% RSLogix 500 project SW2012_BE.RSS, saved by version 12.00.00.00 %
PROJECT "PS8"    % processor: MicroLogix 1400 %

PROGRAM FILES
  LAD 2 "MAIN"  23 rungs  % Calls all system and subsystem routines %
  LAD 3 "CONSTANTS"  50 rungs  % Maintains the system constants %
  LAD 4 "DEFAULTS"  54 rungs  % Manages the system default values %
  LAD 5 "SYS_FAULTS"  45 rungs  % Monitors the system fault conditions %
  LAD 6 "SYSTEM"  71 rungs  % Controls the system %
  LAD 7 "PROCESSING"  17 rungs  % Runs the processing control %
  LAD 8 "MANUAL_CTL"  9 rungs  % Runs the manual valve control %
  LAD 10 "PURIFY"  37 rungs  % Operates the purify control %
  LAD 11 "REGEN"  79 rungs  % Operates the regen control %
  LAD 12 "REGEN_FLT"  47 rungs  % regen alarms and warnings %
  LAD 17 "BYPASS"  7 rungs  % Controls the bypass %
  LAD 18 "MIX PANEL"  12 rungs
  LAD 20 "ADS_A"  47 rungs  % Controls the Adsorber A %
  LAD 21 "ADS_A_FLT"  17 rungs  % Controls the Adsorber A faults %
  LAD 22 "ADS_B"  47 rungs  % Controld Adsorber B %
  LAD 23 "ADS_B_FLT"  17 rungs  % Controls the Adsorber B faults %
  LAD 24 "PREHEATER"  9 rungs
  LAD 25 "PH_FLT"  15 rungs
  LAD 49 "MODBUS"  37 rungs
  LAD 50 "PLC_FAULT"  2 rungs
  LAD 51 "REVERSE"  9 rungs

DATA FILES
  O0 OUTPUT  24 elements
  I1 INPUT  25 elements
  S2 STATUS  66 elements
  B3 BINARY  4 elements
  T4 TIMER  112 elements
  C5 COUNTER  21 elements
  R6 CONTROL  2 elements
  N7 SYSTEM CFG  120 elements  % Maintains the values that characterize the system %
  F8 FLOAT  3 elements
  N9 CONSTANTS  86 elements  % The collection of system and subsystem constants %
  N10 SYSTEM  30 elements  % Contain the values for system control %
  N11 PROCESS  4 elements  % Contains the values for the processing machine %
  N12 PURIFY  25 elements  % Contains the values required for purify %
  N13 REGEN  31 elements  % Contains the values required for regen %
  N15 MANUAL CTL  5 elements  % Contains the data for the manual valve control %
  N16 ADSORBER_A  22 elements  % Contains the values for Adsorber A %
  N17 ADSORBER_B  22 elements  % Contains the values required for Adsorber B %
  N19 BYPASS  2 elements
  N20 MIX PANEL  7 elements
  N21 NOMEMBCKUP  4 elements
  PD25 PID HEATER  4 elements
  B30 SYSTEM CFG  6 elements
  B31 SYSTEM  18 elements
  B32 PROCESS  1 elements
  B33 PURIFY  2 elements
  B34 REGEN  3 elements
  B35 MANUAL CTL  3 elements
  B38 BYPASS  1 elements
  L52 SERIAL  1 elements
  N64 MODBUS  126 elements
  L65 TOTAL FLOW  1 elements
  MG68   1 elements
  B69   3 elements
  RIX80   1 elements
  N200 STATUS_SYS  1 elements  % HMI System Status %
  L201 STATUS_PUR  1 elements  % HMI Purifier Status  %
  L202 STATUS_GET  3 elements  % HMI Getter Status %
  L203 STATUS_ADS  3 elements  % HMI Adsorber Status %
  F206 FLOAT_PRC  4 elements  % HMI Purify function Float Values %
  N207 STATUS_PRC  7 elements  % HMI Purify Process function status %
  N210 BUZZER  5 elements  % ALARM BUZZER CONTROL %

LADDER 2 "MAIN"    % Calls all system and subsystem routines %
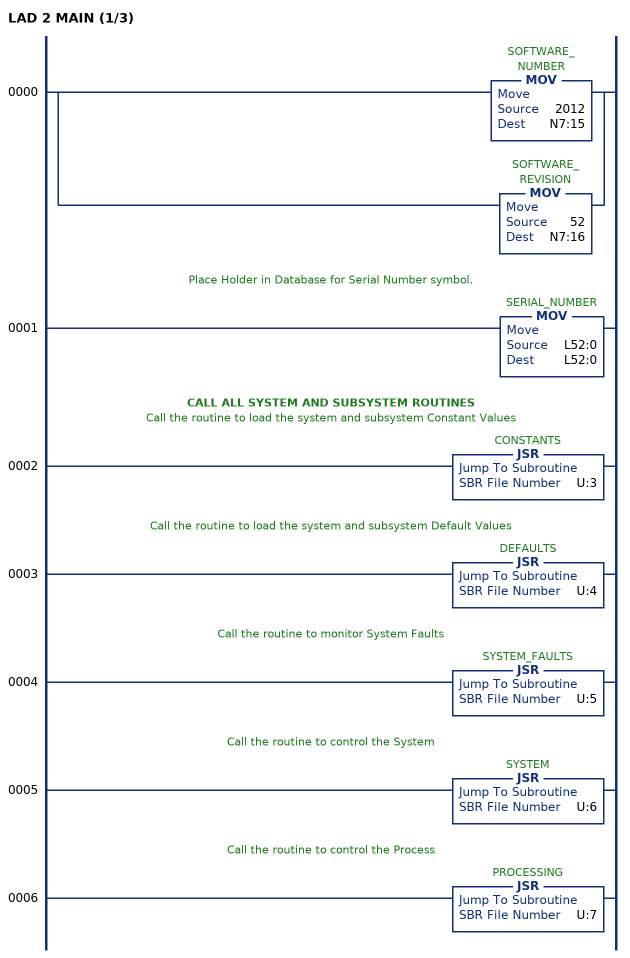
% Rung: 0 %
SOR BST MOV 2012 N7:15 NXB MOV 52 N7:16 BND EOR
%   N7:15  SOFTWARE_NUMBER %
%   N7:16  SOFTWARE_REVISION %
% Rung: 1 %
% Place Holder in Database for Serial Number symbol. %
SOR MOV L52:0 L52:0 EOR
%   L52:0  SERIAL_NUMBER %
% Rung: 2 %
% TITLE: CALL ALL SYSTEM AND SUBSYSTEM ROUTINES %
% Call the routine to load the system and subsystem Constant Values %
SOR JSR U:3 EOR
%   U:3  CONSTANTS %
% Rung: 3 %
% Call the routine to load the system and subsystem Default Values %
SOR JSR U:4 EOR
%   U:4  DEFAULTS %
% Rung: 4 %
% Call the routine to monitor System Faults %
SOR JSR U:5 EOR
%   U:5  SYSTEM_FAULTS %
% Rung: 5 %
% Call the routine to control the System %
SOR JSR U:6 EOR
%   U:6  SYSTEM %
% Rung: 6 %
% Call the routine to control the Process %
SOR JSR U:7 EOR
%   U:7  PROCESSING %

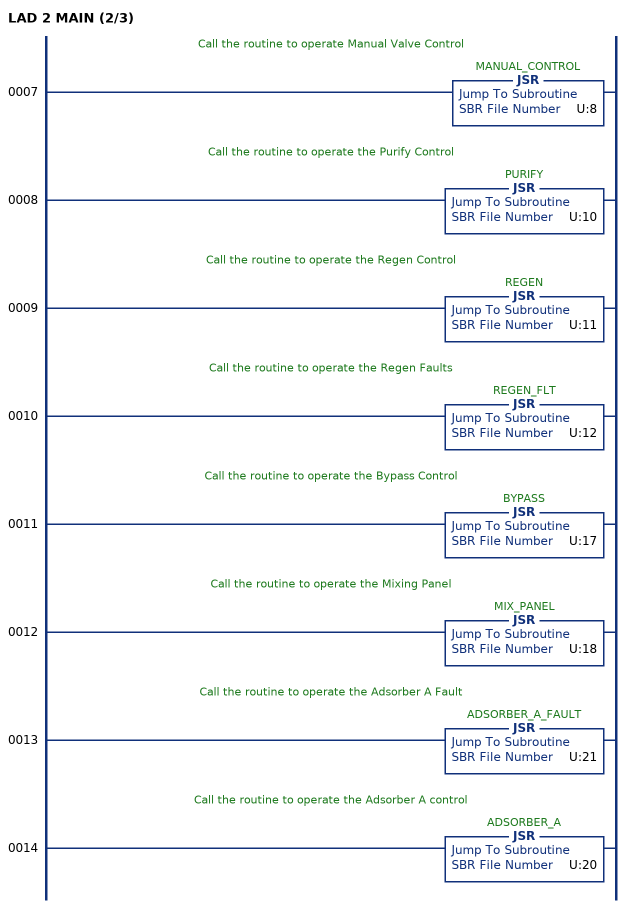
% Rung: 7 %
% Call the routine to operate Manual Valve Control %
SOR JSR U:8 EOR
%   U:8  MANUAL_CONTROL %
% Rung: 8 %
% Call the routine to operate the Purify Control %
SOR JSR U:10 EOR
%   U:10  PURIFY %
% Rung: 9 %
% Call the routine to operate the Regen Control %
SOR JSR U:11 EOR
%   U:11  REGEN %
% Rung: 10 %
% Call the routine to operate the Regen Faults %
SOR JSR U:12 EOR
%   U:12  REGEN_FLT %
% Rung: 11 %
% Call the routine to operate the Bypass Control %
SOR JSR U:17 EOR
%   U:17  BYPASS %
% Rung: 12 %
% Call the routine to operate the Mixing Panel %
SOR JSR U:18 EOR
%   U:18  MIX_PANEL %
% Rung: 13 %
% Call the routine to operate the Adsorber A Fault %
SOR JSR U:21 EOR
%   U:21  ADSORBER_A_FAULT %
% Rung: 14 %
% Call the routine to operate the Adsorber A control %
SOR JSR U:20 EOR
%   U:20  ADSORBER_A %

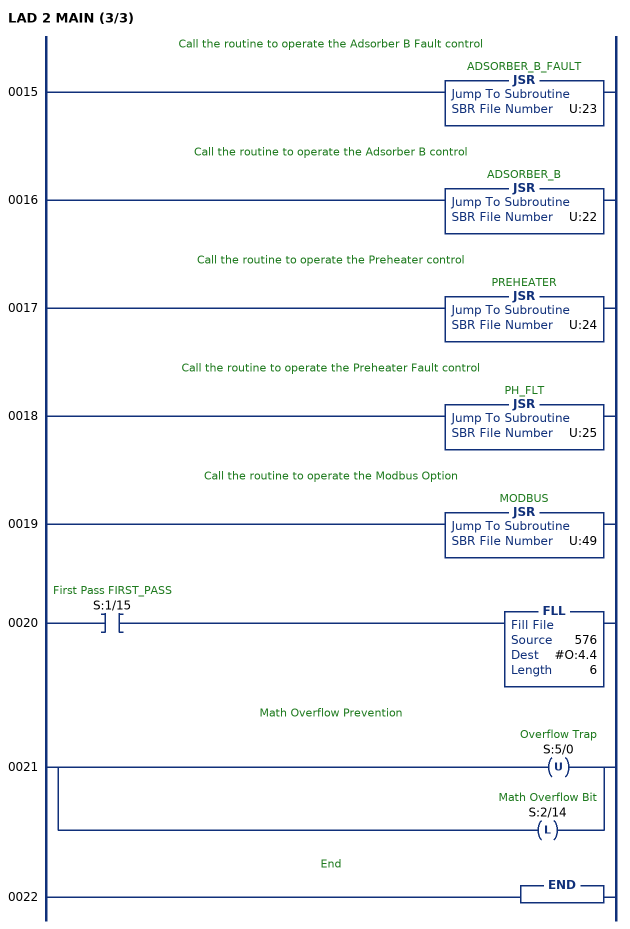
% Rung: 15 %
% Call the routine to operate the Adsorber B Fault control %
SOR JSR U:23 EOR
%   U:23  ADSORBER_B_FAULT %
% Rung: 16 %
% Call the routine to operate the Adsorber B control %
SOR JSR U:22 EOR
%   U:22  ADSORBER_B %
% Rung: 17 %
% Call the routine to operate the Preheater control %
SOR JSR U:24 EOR
%   U:24  PREHEATER %
% Rung: 18 %
% Call the routine to operate the Preheater Fault control %
SOR JSR U:25 EOR
%   U:25  PH_FLT %
% Rung: 19 %
% Call the routine to operate the Modbus Option %
SOR JSR U:49 EOR
%   U:49  MODBUS %
% Rung: 20 %
SOR XIC S:1/15 FLL 576 #O:4.4 6 EOR
%   S:1/15  FIRST_PASS  "First Pass" %
% Rung: 21 %
% Math Overflow Prevention %
SOR BST OTU S:5/0 NXB OTL S:2/14 BND EOR
%   S:5/0  "Overflow Trap" %
%   S:2/14  "Math Overflow Bit" %
% Rung: 22 %
% End %
SOR END EOR

LADDER 3 "CONSTANTS"    % Maintains the system constants %
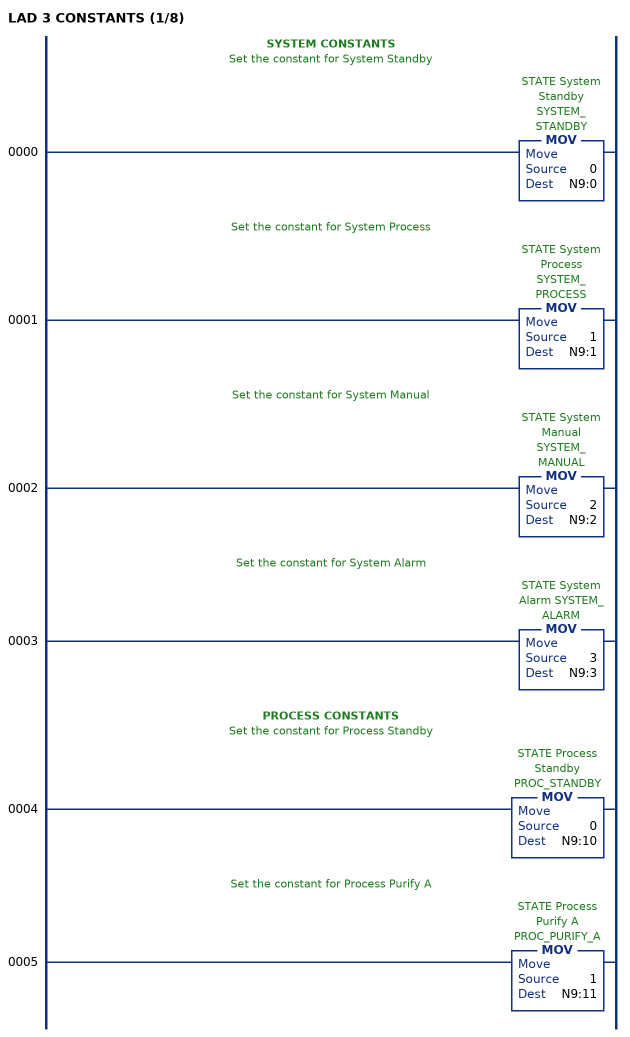
% Rung: 0 %
% TITLE: SYSTEM CONSTANTS %
% Set the constant for System Standby %
SOR MOV 0 N9:0 EOR
%   N9:0  SYSTEM_STANDBY  "STATE System Standby" %
% Rung: 1 %
% Set the constant for System Process %
SOR MOV 1 N9:1 EOR
%   N9:1  SYSTEM_PROCESS  "STATE System Process" %
% Rung: 2 %
% Set the constant for System Manual %
SOR MOV 2 N9:2 EOR
%   N9:2  SYSTEM_MANUAL  "STATE System Manual" %
% Rung: 3 %
% Set the constant for System Alarm %
SOR MOV 3 N9:3 EOR
%   N9:3  SYSTEM_ALARM  "STATE System Alarm" %
% Rung: 4 %
% TITLE: PROCESS CONSTANTS %
% Set the constant for Process Standby %
SOR MOV 0 N9:10 EOR
%   N9:10  PROC_STANDBY  "STATE Process Standby" %
% Rung: 5 %
% Set the constant for Process Purify A %
SOR MOV 1 N9:11 EOR
%   N9:11  PROC_PURIFY_A  "STATE Process Purify A" %

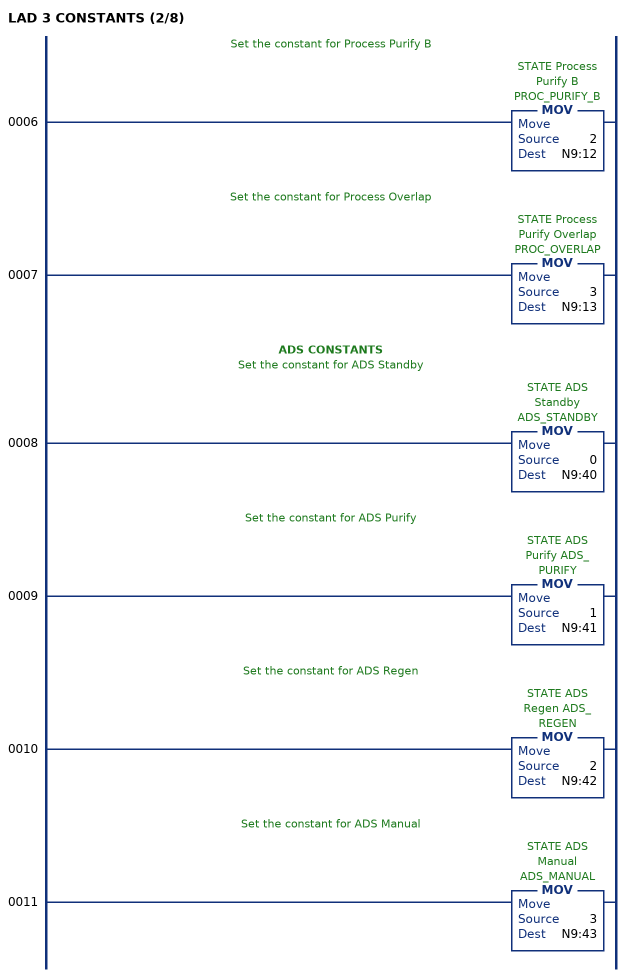
% Rung: 6 %
% Set the constant for Process Purify B %
SOR MOV 2 N9:12 EOR
%   N9:12  PROC_PURIFY_B  "STATE Process Purify B" %
% Rung: 7 %
% Set the constant for Process Overlap %
SOR MOV 3 N9:13 EOR
%   N9:13  PROC_OVERLAP  "STATE Process Purify Overlap" %
% Rung: 8 %
% TITLE: ADS CONSTANTS %
% Set the constant for ADS Standby %
SOR MOV 0 N9:40 EOR
%   N9:40  ADS_STANDBY  "STATE ADS Standby" %
% Rung: 9 %
% Set the constant for ADS Purify %
SOR MOV 1 N9:41 EOR
%   N9:41  ADS_PURIFY  "STATE ADS Purify" %
% Rung: 10 %
% Set the constant for ADS Regen %
SOR MOV 2 N9:42 EOR
%   N9:42  ADS_REGEN  "STATE ADS Regen" %
% Rung: 11 %
% Set the constant for ADS Manual %
SOR MOV 3 N9:43 EOR
%   N9:43  ADS_MANUAL  "STATE ADS Manual" %

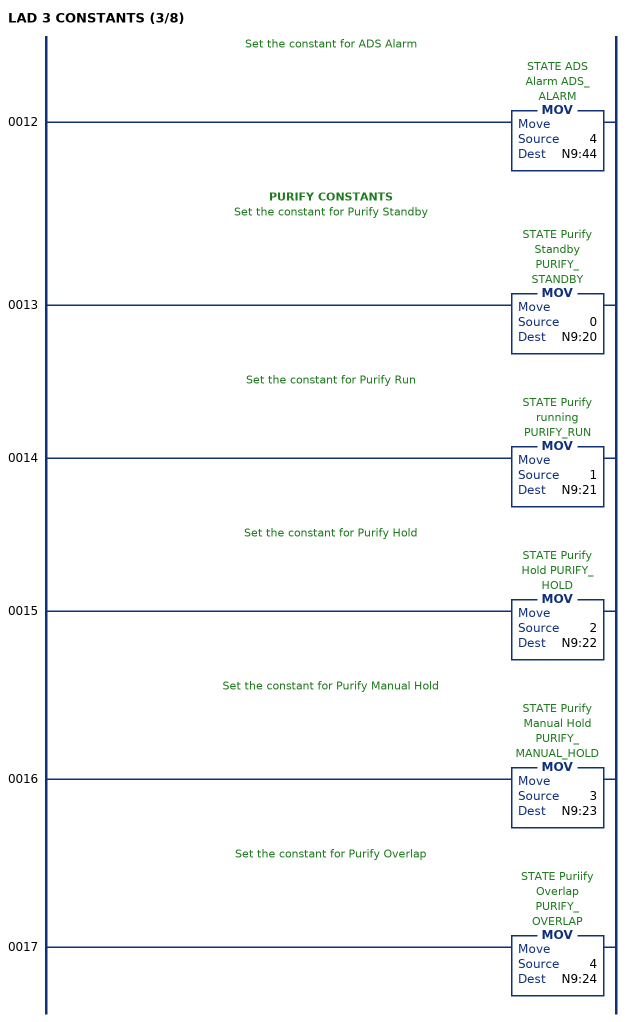
% Rung: 12 %
% Set the constant for ADS Alarm %
SOR MOV 4 N9:44 EOR
%   N9:44  ADS_ALARM  "STATE ADS Alarm" %
% Rung: 13 %
% TITLE: PURIFY CONSTANTS %
% Set the constant for Purify Standby %
SOR MOV 0 N9:20 EOR
%   N9:20  PURIFY_STANDBY  "STATE Purify Standby" %
% Rung: 14 %
% Set the constant for Purify Run %
SOR MOV 1 N9:21 EOR
%   N9:21  PURIFY_RUN  "STATE Purify running" %
% Rung: 15 %
% Set the constant for Purify Hold %
SOR MOV 2 N9:22 EOR
%   N9:22  PURIFY_HOLD  "STATE Purify Hold" %
% Rung: 16 %
% Set the constant for Purify Manual Hold %
SOR MOV 3 N9:23 EOR
%   N9:23  PURIFY_MANUAL_HOLD  "STATE Purify Manual Hold" %
% Rung: 17 %
% Set the constant for Purify Overlap %
SOR MOV 4 N9:24 EOR
%   N9:24  PURIFY_OVERLAP  "STATE Puriify Overlap" %

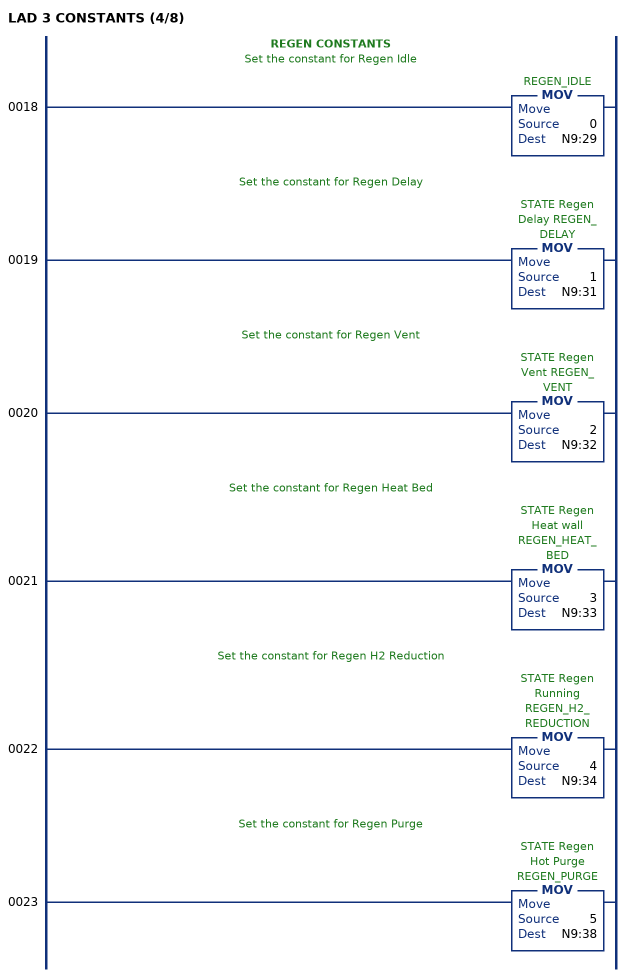
% Rung: 18 %
% TITLE: REGEN CONSTANTS %
% Set the constant for Regen Idle %
SOR MOV 0 N9:29 EOR
%   N9:29  REGEN_IDLE %
% Rung: 19 %
% Set the constant for Regen Delay %
SOR MOV 1 N9:31 EOR
%   N9:31  REGEN_DELAY  "STATE Regen Delay" %
% Rung: 20 %
% Set the constant for Regen Vent %
SOR MOV 2 N9:32 EOR
%   N9:32  REGEN_VENT  "STATE Regen Vent" %
% Rung: 21 %
% Set the constant for Regen Heat Bed %
SOR MOV 3 N9:33 EOR
%   N9:33  REGEN_HEAT_BED  "STATE Regen Heat wall" %
% Rung: 22 %
% Set the constant for Regen H2 Reduction %
SOR MOV 4 N9:34 EOR
%   N9:34  REGEN_H2_REDUCTION  "STATE Regen Running" %
% Rung: 23 %
% Set the constant for Regen Purge %
SOR MOV 5 N9:38 EOR
%   N9:38  REGEN_PURGE  "STATE Regen Hot Purge" %

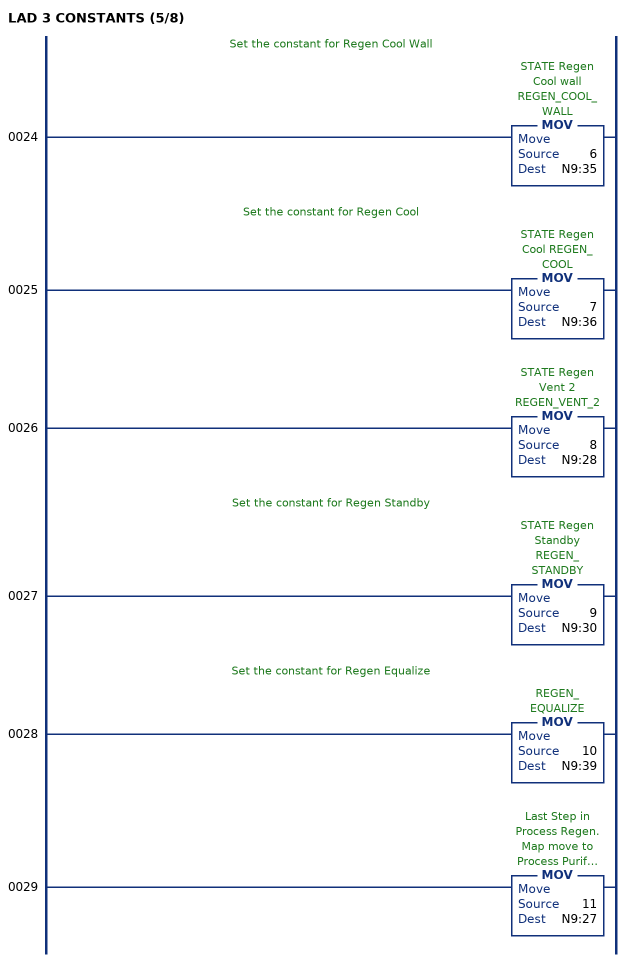
% Rung: 24 %
% Set the constant for Regen Cool Wall %
SOR MOV 6 N9:35 EOR
%   N9:35  REGEN_COOL_WALL  "STATE Regen Cool wall" %
% Rung: 25 %
% Set the constant for Regen Cool %
SOR MOV 7 N9:36 EOR
%   N9:36  REGEN_COOL  "STATE Regen Cool" %
% Rung: 26 %
SOR MOV 8 N9:28 EOR
%   N9:28  REGEN_VENT_2  "STATE Regen Vent 2" %
% Rung: 27 %
% Set the constant for Regen Standby %
SOR MOV 9 N9:30 EOR
%   N9:30  REGEN_STANDBY  "STATE Regen Standby" %
% Rung: 28 %
% Set the constant for Regen Equalize %
SOR MOV 10 N9:39 EOR
%   N9:39  REGEN_EQUALIZE %
% Rung: 29 %
SOR MOV 11 N9:27 EOR
%   N9:27  REGEN_PUR_OVERLAP  "Last Step in Process Regen. Map move to Process Purify overlap." %

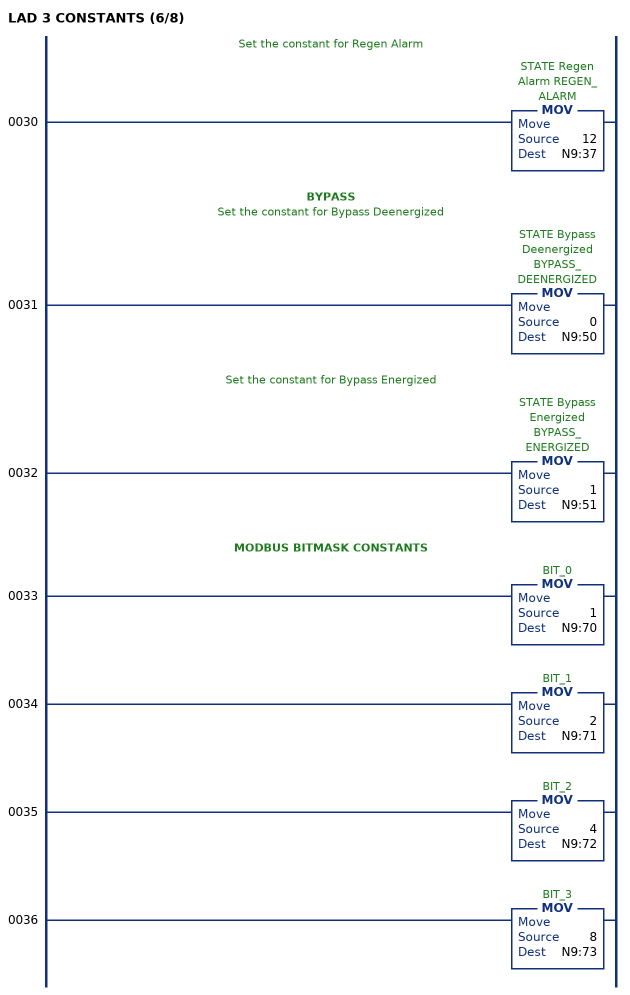
% Rung: 30 %
% Set the constant for Regen Alarm %
SOR MOV 12 N9:37 EOR
%   N9:37  REGEN_ALARM  "STATE Regen Alarm" %
% Rung: 31 %
% TITLE: BYPASS %
% Set the constant for Bypass Deenergized %
SOR MOV 0 N9:50 EOR
%   N9:50  BYPASS_DEENERGIZED  "STATE Bypass Deenergized" %
% Rung: 32 %
% Set the constant for Bypass Energized %
SOR MOV 1 N9:51 EOR
%   N9:51  BYPASS_ENERGIZED  "STATE Bypass Energized" %
% Rung: 33 %
% TITLE: MODBUS BITMASK CONSTANTS %
SOR MOV 1 N9:70 EOR
%   N9:70  BIT_0 %
% Rung: 34 %
SOR MOV 2 N9:71 EOR
%   N9:71  BIT_1 %
% Rung: 35 %
SOR MOV 4 N9:72 EOR
%   N9:72  BIT_2 %
% Rung: 36 %
SOR MOV 8 N9:73 EOR
%   N9:73  BIT_3 %

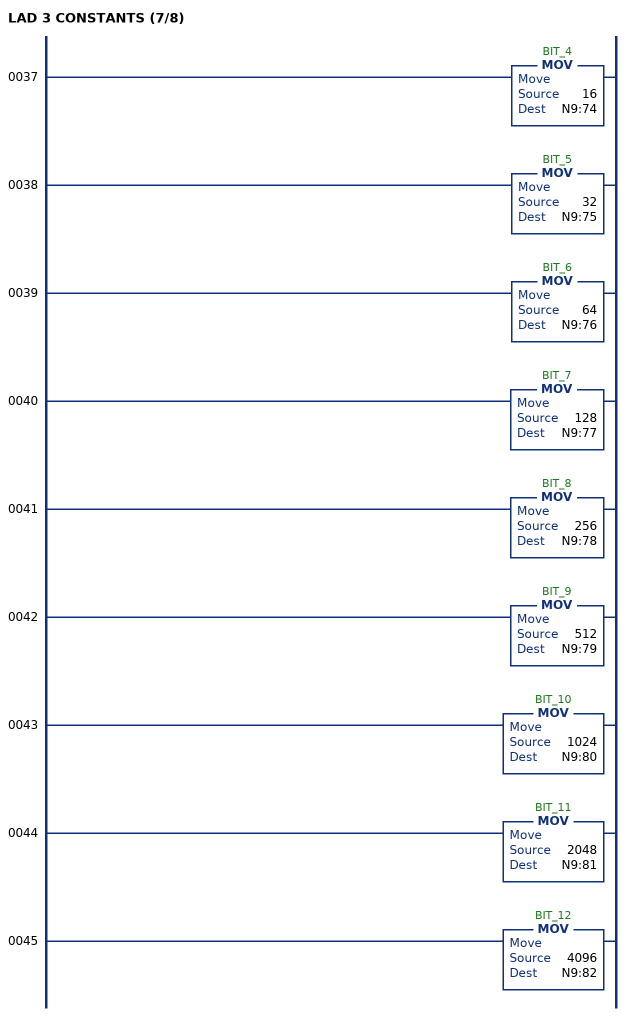
% Rung: 37 %
SOR MOV 16 N9:74 EOR
%   N9:74  BIT_4 %
% Rung: 38 %
SOR MOV 32 N9:75 EOR
%   N9:75  BIT_5 %
% Rung: 39 %
SOR MOV 64 N9:76 EOR
%   N9:76  BIT_6 %
% Rung: 40 %
SOR MOV 128 N9:77 EOR
%   N9:77  BIT_7 %
% Rung: 41 %
SOR MOV 256 N9:78 EOR
%   N9:78  BIT_8 %
% Rung: 42 %
SOR MOV 512 N9:79 EOR
%   N9:79  BIT_9 %
% Rung: 43 %
SOR MOV 1024 N9:80 EOR
%   N9:80  BIT_10 %
% Rung: 44 %
SOR MOV 2048 N9:81 EOR
%   N9:81  BIT_11 %
% Rung: 45 %
SOR MOV 4096 N9:82 EOR
%   N9:82  BIT_12 %

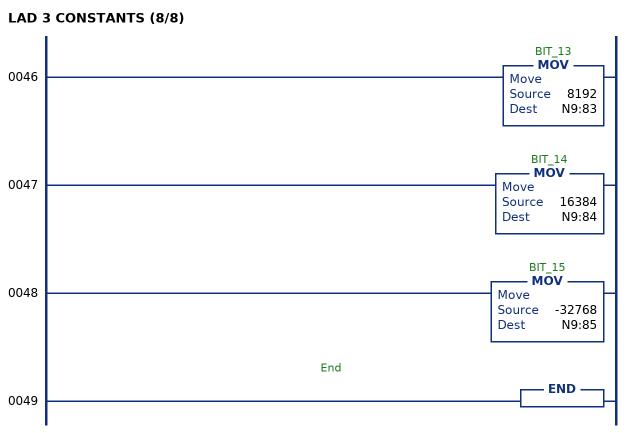
% Rung: 46 %
SOR MOV 8192 N9:83 EOR
%   N9:83  BIT_13 %
% Rung: 47 %
SOR MOV 16384 N9:84 EOR
%   N9:84  BIT_14 %
% Rung: 48 %
SOR MOV -32768 N9:85 EOR
%   N9:85  BIT_15 %
% Rung: 49 %
% End %
SOR END EOR

LADDER 4 "DEFAULTS"    % Manages the system default values %
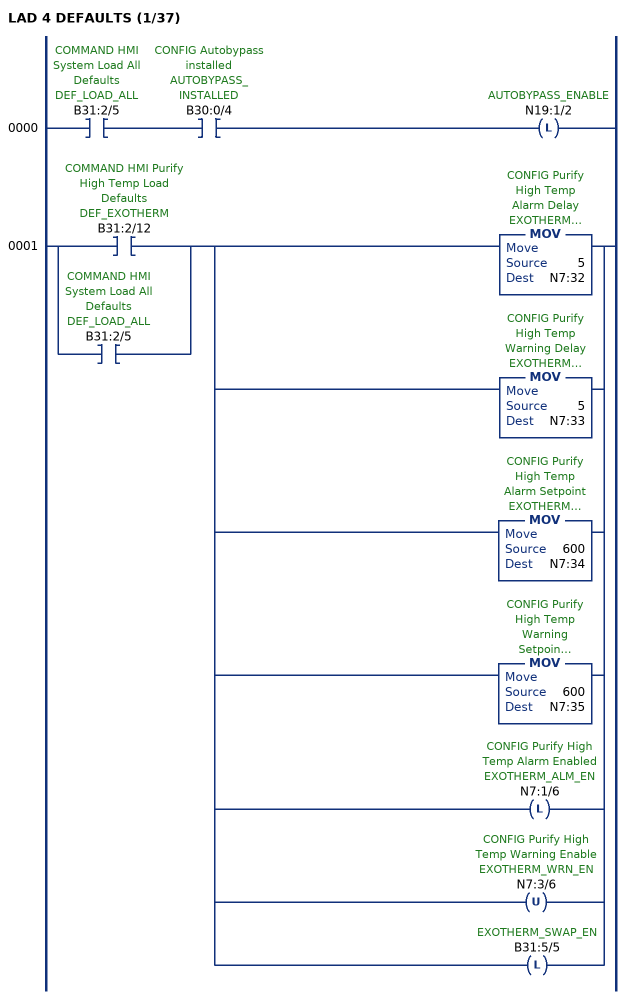
% Rung: 0 %
SOR XIC B31:2/5 XIC B30:0/4 OTL N19:1/2 EOR
%   B31:2/5  DEF_LOAD_ALL  "COMMAND HMI System Load All Defaults" %
%   B30:0/4  AUTOBYPASS_INSTALLED  "CONFIG Autobypass installed" %
%   N19:1/2  AUTOBYPASS_ENABLE %
% Rung: 1 %
SOR BST XIC B31:2/12 NXB XIC B31:2/5 BND BST MOV 5 N7:32 NXB MOV 5 N7:33 NXB MOV 600 N7:34 NXB MOV 600 N7:35 NXB OTL N7:1/6 NXB OTU N7:3/6 NXB OTL B31:5/5 BND EOR
%   B31:2/12  DEF_EXOTHERM  "COMMAND HMI Purify High Temp Load Defaults" %
%   B31:2/5  DEF_LOAD_ALL  "COMMAND HMI System Load All Defaults" %
%   N7:32  EXOTHERM_ALM_DLY  "CONFIG Purify High Temp Alarm Delay" %
%   N7:33  EXOTHERM_WRN_DLY  "CONFIG Purify High Temp Warning Delay" %
%   N7:34  EXOTHERM_ALM_SP  "CONFIG Purify High Temp Alarm Setpoint" %
%   N7:35  EXOTHERM_WRN_SP  "CONFIG Purify High Temp Warning Setpoint" %
%   N7:1/6  EXOTHERM_ALM_EN  "CONFIG Purify High Temp Alarm Enabled" %
%   N7:3/6  EXOTHERM_WRN_EN  "CONFIG Purify High Temp Warning Enable" %
%   B31:5/5  EXOTHERM_SWAP_EN %

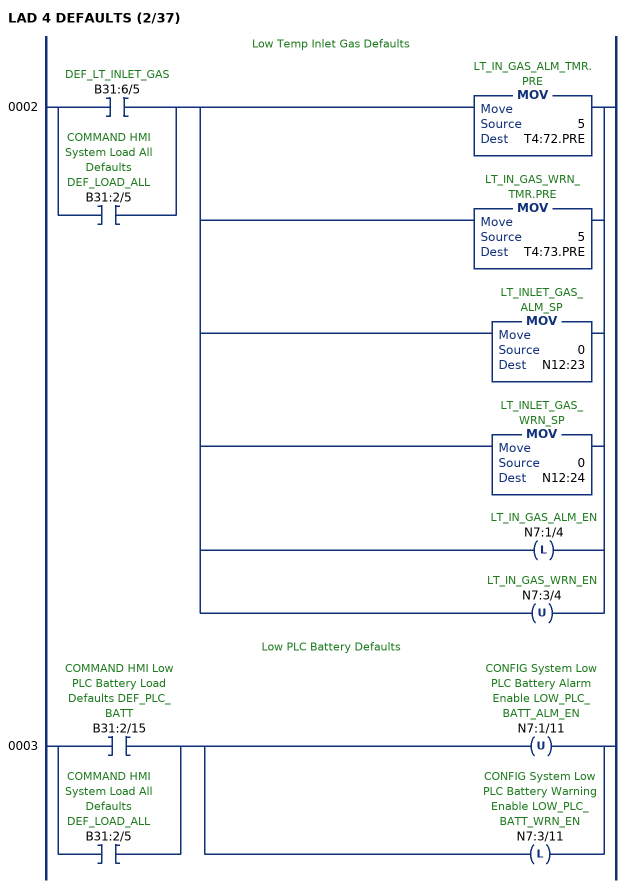
% Rung: 2 %
% Low Temp Inlet Gas Defaults %
SOR BST XIC B31:6/5 NXB XIC B31:2/5 BND BST MOV 5 T4:72.PRE NXB MOV 5 T4:73.PRE NXB MOV 0 N12:23 NXB MOV 0 N12:24 NXB OTL N7:1/4 NXB OTU N7:3/4 BND EOR
%   B31:6/5  DEF_LT_INLET_GAS %
%   B31:2/5  DEF_LOAD_ALL  "COMMAND HMI System Load All Defaults" %
%   T4:72  LT_IN_GAS_ALM_TMR %
%   T4:73  LT_IN_GAS_WRN_TMR %
%   N12:23  LT_INLET_GAS_ALM_SP %
%   N12:24  LT_INLET_GAS_WRN_SP %
%   N7:1/4  LT_IN_GAS_ALM_EN %
%   N7:3/4  LT_IN_GAS_WRN_EN %
% Rung: 3 %
% Low PLC Battery Defaults %
SOR BST XIC B31:2/15 NXB XIC B31:2/5 BND BST OTU N7:1/11 NXB OTL N7:3/11 BND EOR
%   B31:2/15  DEF_PLC_BATT  "COMMAND HMI Low PLC Battery Load Defaults" %
%   B31:2/5  DEF_LOAD_ALL  "COMMAND HMI System Load All Defaults" %
%   N7:1/11  LOW_PLC_BATT_ALM_EN  "CONFIG System Low PLC Battery Alarm Enable" %
%   N7:3/11  LOW_PLC_BATT_WRN_EN  "CONFIG System Low PLC Battery Warning Enable" %

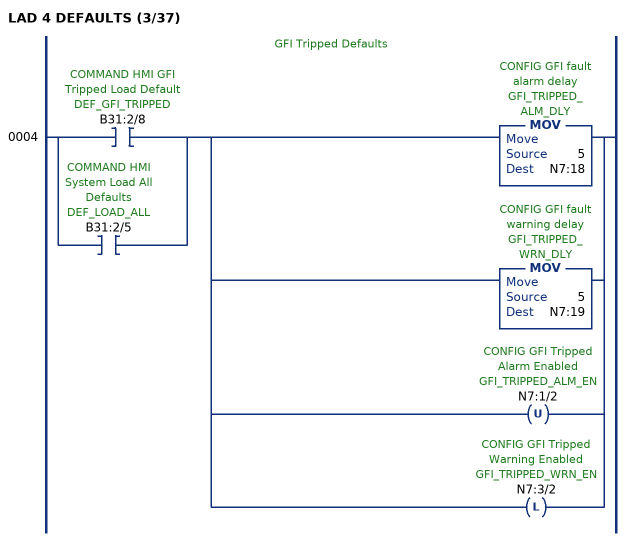
% Rung: 4 %
% GFI Tripped Defaults %
SOR BST XIC B31:2/8 NXB XIC B31:2/5 BND BST MOV 5 N7:18 NXB MOV 5 N7:19 NXB OTU N7:1/2 NXB OTL N7:3/2 BND EOR
%   B31:2/8  DEF_GFI_TRIPPED  "COMMAND HMI GFI Tripped Load Default" %
%   B31:2/5  DEF_LOAD_ALL  "COMMAND HMI System Load All Defaults" %
%   N7:18  GFI_TRIPPED_ALM_DLY  "CONFIG GFI fault alarm delay" %
%   N7:19  GFI_TRIPPED_WRN_DLY  "CONFIG GFI fault warning delay" %
%   N7:1/2  GFI_TRIPPED_ALM_EN  "CONFIG GFI Tripped Alarm Enabled" %
%   N7:3/2  GFI_TRIPPED_WRN_EN  "CONFIG GFI Tripped Warning Enabled" %

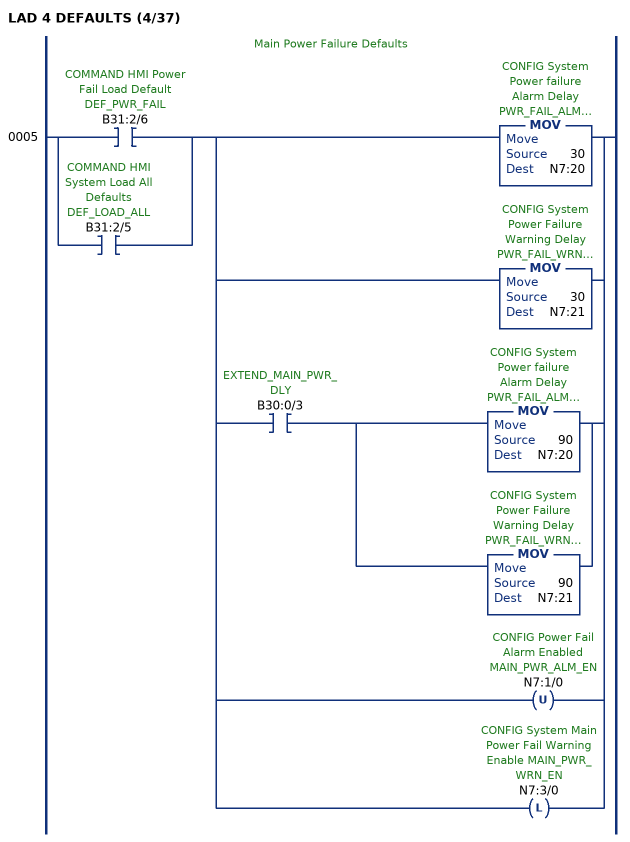
% Rung: 5 %
% Main Power Failure Defaults %
SOR BST XIC B31:2/6 NXB XIC B31:2/5 BND BST MOV 30 N7:20 NXB MOV 30 N7:21 NXB XIC B30:0/3 BST MOV 90 N7:20 NXB MOV 90 N7:21 BND NXB OTU N7:1/0 NXB OTL N7:3/0 BND EOR
%   B31:2/6  DEF_PWR_FAIL  "COMMAND HMI Power Fail Load Default" %
%   B31:2/5  DEF_LOAD_ALL  "COMMAND HMI System Load All Defaults" %
%   N7:20  PWR_FAIL_ALM_DELAY  "CONFIG System Power failure Alarm Delay" %
%   N7:21  PWR_FAIL_WRN_DELAY  "CONFIG System Power Failure Warning Delay" %
%   B30:0/3  EXTEND_MAIN_PWR_DLY %
%   N7:1/0  MAIN_PWR_ALM_EN  "CONFIG Power Fail Alarm Enabled" %
%   N7:3/0  MAIN_PWR_WRN_EN  "CONFIG System Main Power Fail Warning Enable" %

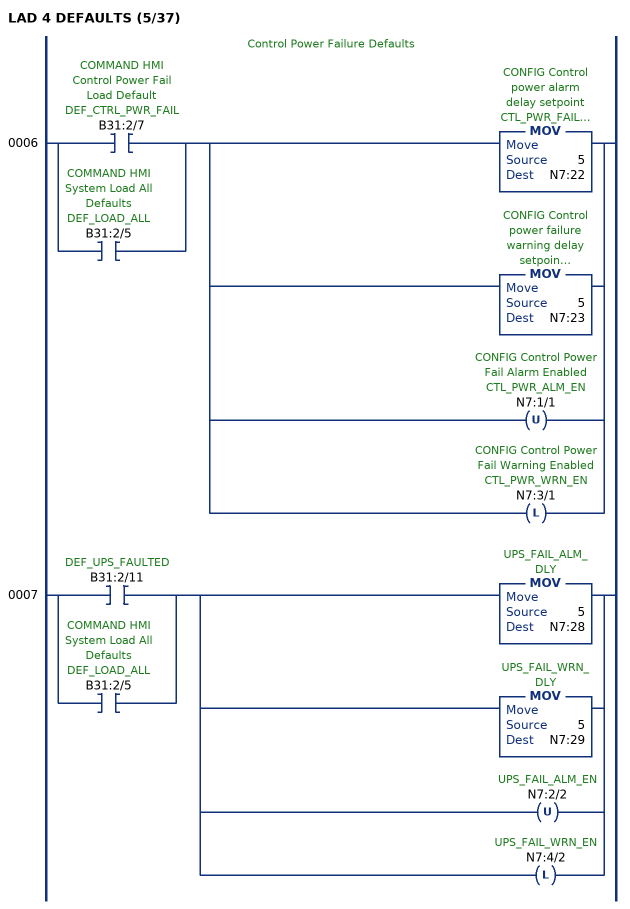
% Rung: 6 %
% Control Power Failure Defaults %
SOR BST XIC B31:2/7 NXB XIC B31:2/5 BND BST MOV 5 N7:22 NXB MOV 5 N7:23 NXB OTU N7:1/1 NXB OTL N7:3/1 BND EOR
%   B31:2/7  DEF_CTRL_PWR_FAIL  "COMMAND HMI Control Power Fail Load Default" %
%   B31:2/5  DEF_LOAD_ALL  "COMMAND HMI System Load All Defaults" %
%   N7:22  CTL_PWR_FAIL_ALM_DLY  "CONFIG Control power alarm delay setpoint" %
%   N7:23  CTL_PWR_FAIL_WRN_DLY  "CONFIG Control power failure warning delay setpoint" %
%   N7:1/1  CTL_PWR_ALM_EN  "CONFIG Control Power Fail Alarm Enabled" %
%   N7:3/1  CTL_PWR_WRN_EN  "CONFIG Control Power Fail Warning Enabled" %
% Rung: 7 %
SOR BST XIC B31:2/11 NXB XIC B31:2/5 BND BST MOV 5 N7:28 NXB MOV 5 N7:29 NXB OTU N7:2/2 NXB OTL N7:4/2 BND EOR
%   B31:2/11  DEF_UPS_FAULTED %
%   B31:2/5  DEF_LOAD_ALL  "COMMAND HMI System Load All Defaults" %
%   N7:28  UPS_FAIL_ALM_DLY %
%   N7:29  UPS_FAIL_WRN_DLY %
%   N7:2/2  UPS_FAIL_ALM_EN %
%   N7:4/2  UPS_FAIL_WRN_EN %

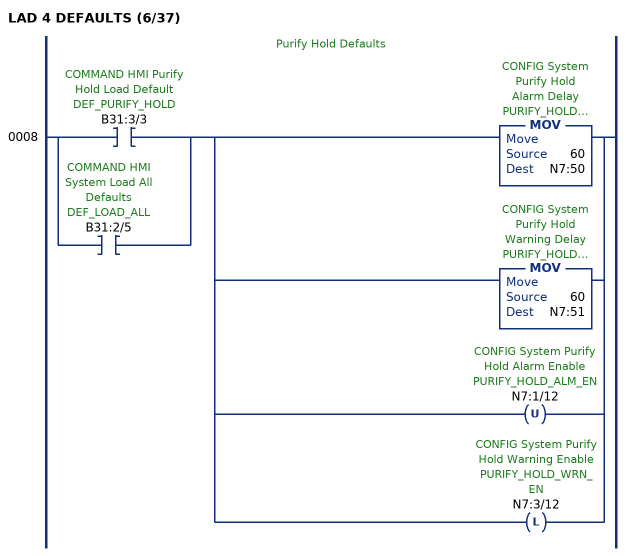
% Rung: 8 %
% Purify Hold Defaults %
SOR BST XIC B31:3/3 NXB XIC B31:2/5 BND BST MOV 60 N7:50 NXB MOV 60 N7:51 NXB OTU N7:1/12 NXB OTL N7:3/12 BND EOR
%   B31:3/3  DEF_PURIFY_HOLD  "COMMAND HMI Purify Hold Load Default" %
%   B31:2/5  DEF_LOAD_ALL  "COMMAND HMI System Load All Defaults" %
%   N7:50  PURIFY_HOLD_ALM_DLY  "CONFIG System Purify Hold Alarm Delay" %
%   N7:51  PURIFY_HOLD_WRN_DLY  "CONFIG System Purify Hold Warning Delay" %
%   N7:1/12  PURIFY_HOLD_ALM_EN  "CONFIG System Purify Hold Alarm Enable" %
%   N7:3/12  PURIFY_HOLD_WRN_EN  "CONFIG System Purify Hold Warning Enable" %

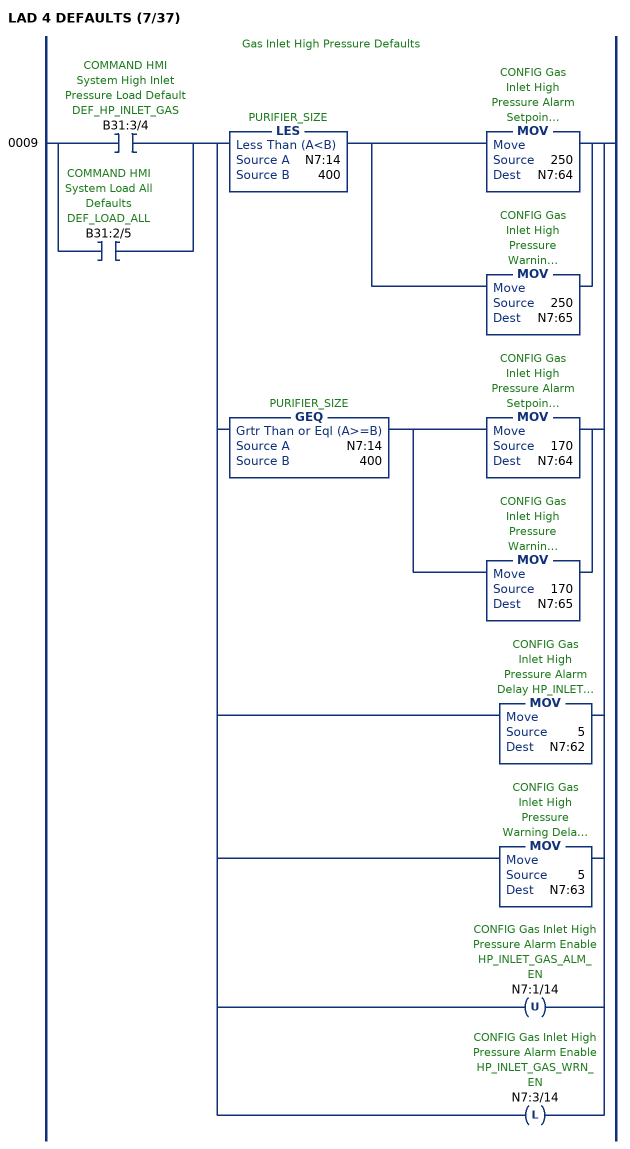
% Rung: 9 %
% Gas Inlet High Pressure Defaults %
SOR BST XIC B31:3/4 NXB XIC B31:2/5 BND BST LES N7:14 400 BST MOV 250 N7:64 NXB MOV 250 N7:65 BND NXB GEQ N7:14 400 BST MOV 170 N7:64 NXB MOV 170 N7:65 BND NXB MOV 5 N7:62 NXB MOV 5 N7:63 NXB OTU N7:1/14 NXB OTL N7:3/14 BND EOR
%   B31:3/4  DEF_HP_INLET_GAS  "COMMAND HMI System High Inlet Pressure Load Default" %
%   B31:2/5  DEF_LOAD_ALL  "COMMAND HMI System Load All Defaults" %
%   N7:14  PURIFIER_SIZE %
%   N7:64  HP_INLET_GAS_ALM_SP  "CONFIG Gas Inlet High Pressure Alarm Setpoint" %
%   N7:65  HP_INLET_GAS_WRN_SP  "CONFIG Gas Inlet High Pressure Warning Setpoint" %
%   N7:62  HP_INLET_GAS_ALM_DLY  "CONFIG Gas Inlet High Pressure Alarm Delay" %
%   N7:63  HP_INLET_GAS_WRN_DLY  "CONFIG Gas Inlet High Pressure Warning Delay" %
%   N7:1/14  HP_INLET_GAS_ALM_EN  "CONFIG Gas Inlet High Pressure Alarm Enable" %
%   N7:3/14  HP_INLET_GAS_WRN_EN  "CONFIG Gas Inlet High Pressure Alarm Enable" %

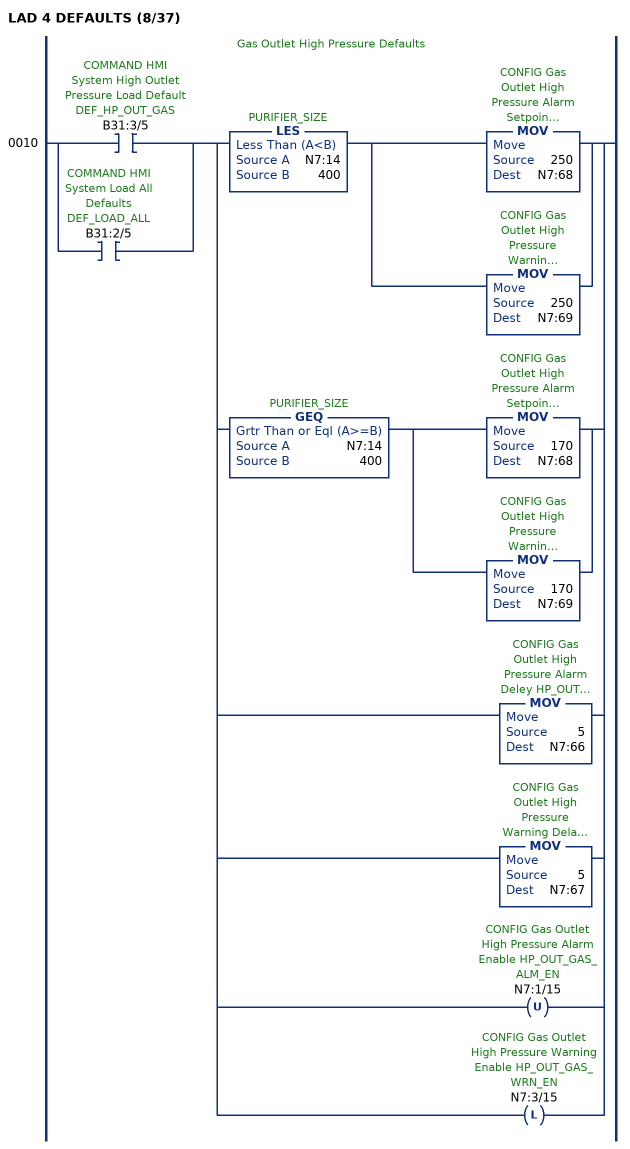
% Rung: 10 %
% Gas Outlet High Pressure Defaults %
SOR BST XIC B31:3/5 NXB XIC B31:2/5 BND BST LES N7:14 400 BST MOV 250 N7:68 NXB MOV 250 N7:69 BND NXB GEQ N7:14 400 BST MOV 170 N7:68 NXB MOV 170 N7:69 BND NXB MOV 5 N7:66 NXB MOV 5 N7:67 NXB OTU N7:1/15 NXB OTL N7:3/15 BND EOR
%   B31:3/5  DEF_HP_OUT_GAS  "COMMAND HMI System High Outlet Pressure Load Default" %
%   B31:2/5  DEF_LOAD_ALL  "COMMAND HMI System Load All Defaults" %
%   N7:14  PURIFIER_SIZE %
%   N7:68  HP_OUT_GAS_ALM_SP  "CONFIG Gas Outlet High Pressure Alarm Setpoint" %
%   N7:69  HP_OUT_GAS_WRN_SP  "CONFIG Gas Outlet High Pressure Warning Setpoint" %
%   N7:66  HP_OUT_GAS_ALM_DLY  "CONFIG Gas Outlet High Pressure Alarm Deley" %
%   N7:67  HP_OUT_GAS_WRN_DLY  "CONFIG Gas Outlet High Pressure Warning Delay" %
%   N7:1/15  HP_OUT_GAS_ALM_EN  "CONFIG Gas Outlet High Pressure Alarm Enable" %
%   N7:3/15  HP_OUT_GAS_WRN_EN  "CONFIG Gas Outlet High Pressure Warning Enable" %

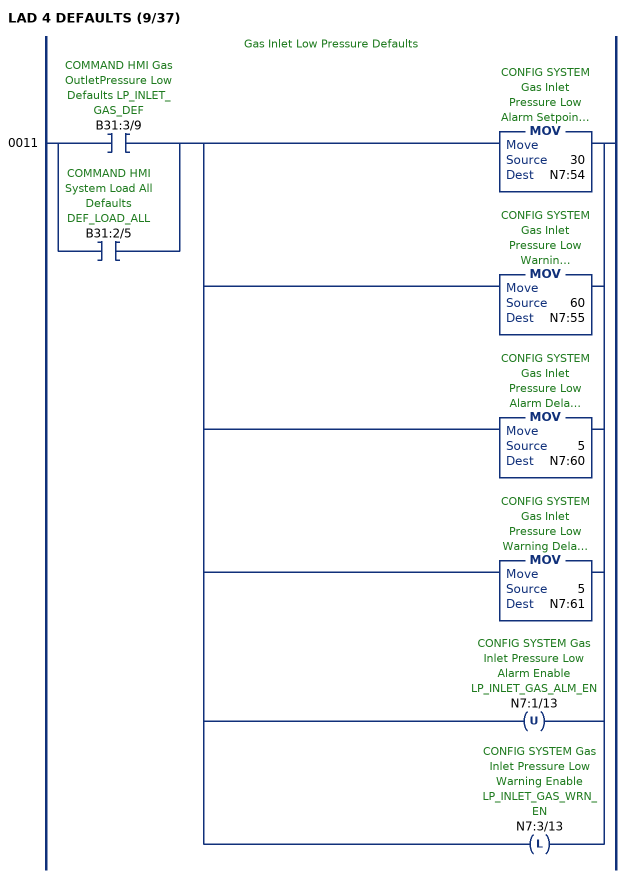
% Rung: 11 %
% Gas Inlet Low Pressure Defaults %
SOR BST XIC B31:3/9 NXB XIC B31:2/5 BND BST MOV 30 N7:54 NXB MOV 60 N7:55 NXB MOV 5 N7:60 NXB MOV 5 N7:61 NXB OTU N7:1/13 NXB OTL N7:3/13 BND EOR
%   B31:3/9  LP_INLET_GAS_DEF  "COMMAND HMI Gas OutletPressure Low Defaults" %
%   B31:2/5  DEF_LOAD_ALL  "COMMAND HMI System Load All Defaults" %
%   N7:54  LP_INLET_GAS_ALM_SP  "CONFIG SYSTEM Gas Inlet Pressure Low Alarm Setpoint" %
%   N7:55  LP_INLET_GAS_WRN_SP  "CONFIG SYSTEM Gas Inlet Pressure Low Warning Setpoint" %
%   N7:60  LP_INLET_GAS_ALM_DLY  "CONFIG SYSTEM Gas Inlet Pressure Low Alarm Delay" %
%   N7:61  LP_INLET_GAS_WRN_DLY  "CONFIG SYSTEM Gas Inlet Pressure Low Warning Delay" %
%   N7:1/13  LP_INLET_GAS_ALM_EN  "CONFIG SYSTEM Gas Inlet Pressure Low Alarm Enable" %
%   N7:3/13  LP_INLET_GAS_WRN_EN  "CONFIG SYSTEM Gas Inlet Pressure Low Warning Enable" %

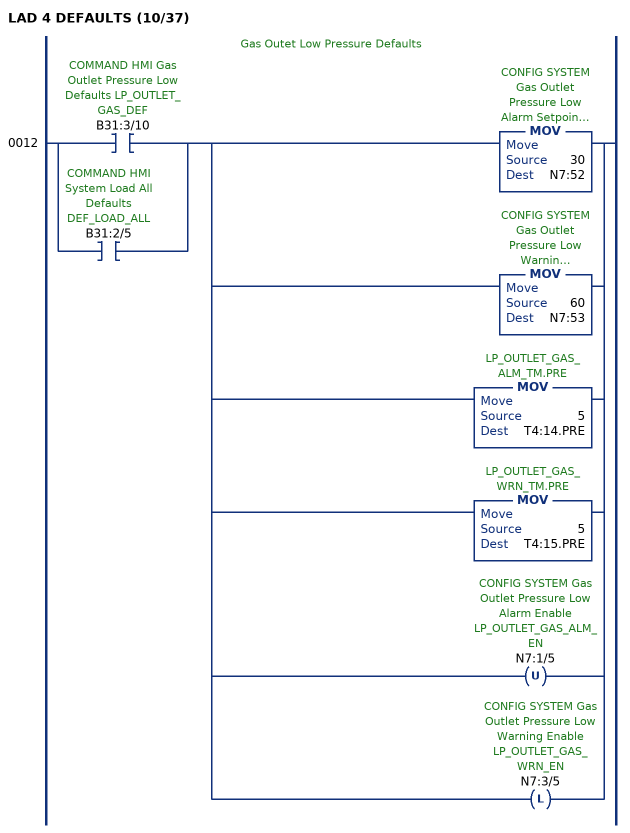
% Rung: 12 %
% Gas Outet Low Pressure Defaults %
SOR BST XIC B31:3/10 NXB XIC B31:2/5 BND BST MOV 30 N7:52 NXB MOV 60 N7:53 NXB MOV 5 T4:14.PRE NXB MOV 5 T4:15.PRE NXB OTU N7:1/5 NXB OTL N7:3/5 BND EOR
%   B31:3/10  LP_OUTLET_GAS_DEF  "COMMAND HMI Gas Outlet Pressure Low Defaults" %
%   B31:2/5  DEF_LOAD_ALL  "COMMAND HMI System Load All Defaults" %
%   N7:52  LP_OUTLET_GAS_ALM_SP  "CONFIG SYSTEM Gas Outlet Pressure Low Alarm Setpoint" %
%   N7:53  LP_OUTLET_GAS_WRN_SP  "CONFIG SYSTEM Gas Outlet Pressure Low Warning Setpoint" %
%   T4:14  LP_OUTLET_GAS_ALM_TM %
%   T4:15  LP_OUTLET_GAS_WRN_TM %
%   N7:1/5  LP_OUTLET_GAS_ALM_EN  "CONFIG SYSTEM Gas Outlet Pressure Low Alarm Enable" %
%   N7:3/5  LP_OUTLET_GAS_WRN_EN  "CONFIG SYSTEM Gas Outlet Pressure Low Warning Enable" %

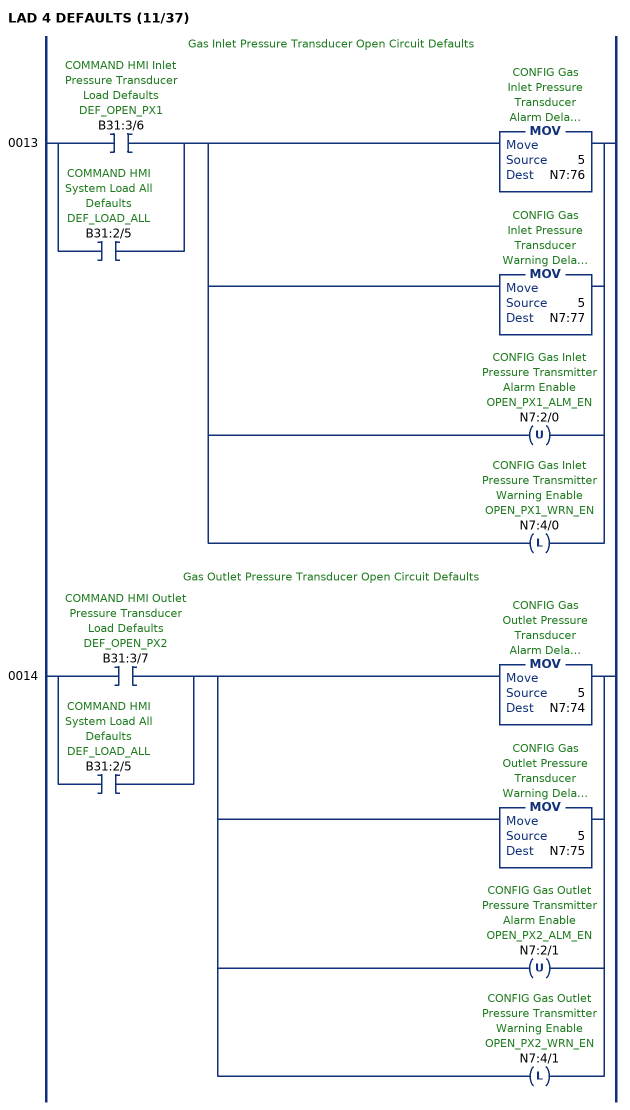
% Rung: 13 %
% Gas Inlet Pressure Transducer Open Circuit Defaults %
SOR BST XIC B31:3/6 NXB XIC B31:2/5 BND BST MOV 5 N7:76 NXB MOV 5 N7:77 NXB OTU N7:2/0 NXB OTL N7:4/0 BND EOR
%   B31:3/6  DEF_OPEN_PX1  "COMMAND HMI Inlet Pressure Transducer Load Defaults" %
%   B31:2/5  DEF_LOAD_ALL  "COMMAND HMI System Load All Defaults" %
%   N7:76  OPEN_PX1_ALM_DLY  "CONFIG Gas Inlet Pressure Transducer Alarm Delay" %
%   N7:77  OPEN_PX1_WRN_DLY  "CONFIG Gas Inlet Pressure Transducer Warning Delay" %
%   N7:2/0  OPEN_PX1_ALM_EN  "CONFIG Gas Inlet Pressure Transmitter Alarm Enable" %
%   N7:4/0  OPEN_PX1_WRN_EN  "CONFIG Gas Inlet Pressure Transmitter Warning Enable" %
% Rung: 14 %
% Gas Outlet Pressure Transducer Open Circuit Defaults %
SOR BST XIC B31:3/7 NXB XIC B31:2/5 BND BST MOV 5 N7:74 NXB MOV 5 N7:75 NXB OTU N7:2/1 NXB OTL N7:4/1 BND EOR
%   B31:3/7  DEF_OPEN_PX2  "COMMAND HMI Outlet Pressure Transducer Load Defaults" %
%   B31:2/5  DEF_LOAD_ALL  "COMMAND HMI System Load All Defaults" %
%   N7:74  OPEN_PX2_ALM_DLY  "CONFIG Gas Outlet Pressure Transducer Alarm Delay" %
%   N7:75  OPEN_PX2_WRN_DLY  "CONFIG Gas Outlet Pressure Transducer Warning Delay" %
%   N7:2/1  OPEN_PX2_ALM_EN  "CONFIG Gas Outlet Pressure Transmitter Alarm Enable" %
%   N7:4/1  OPEN_PX2_WRN_EN  "CONFIG Gas Outlet Pressure Transmitter Warning Enable" %

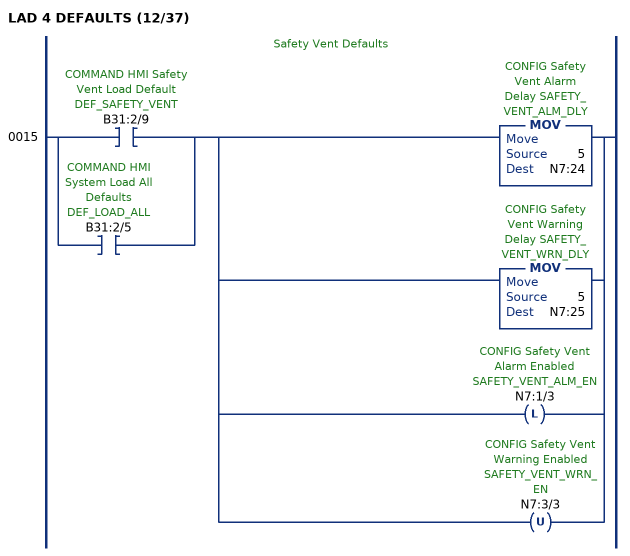
% Rung: 15 %
% Safety Vent Defaults %
SOR BST XIC B31:2/9 NXB XIC B31:2/5 BND BST MOV 5 N7:24 NXB MOV 5 N7:25 NXB OTL N7:1/3 NXB OTU N7:3/3 BND EOR
%   B31:2/9  DEF_SAFETY_VENT  "COMMAND HMI Safety Vent Load Default" %
%   B31:2/5  DEF_LOAD_ALL  "COMMAND HMI System Load All Defaults" %
%   N7:24  SAFETY_VENT_ALM_DLY  "CONFIG Safety Vent Alarm Delay" %
%   N7:25  SAFETY_VENT_WRN_DLY  "CONFIG Safety Vent Warning Delay" %
%   N7:1/3  SAFETY_VENT_ALM_EN  "CONFIG Safety Vent Alarm Enabled" %
%   N7:3/3  SAFETY_VENT_WRN_EN  "CONFIG Safety Vent Warning Enabled" %

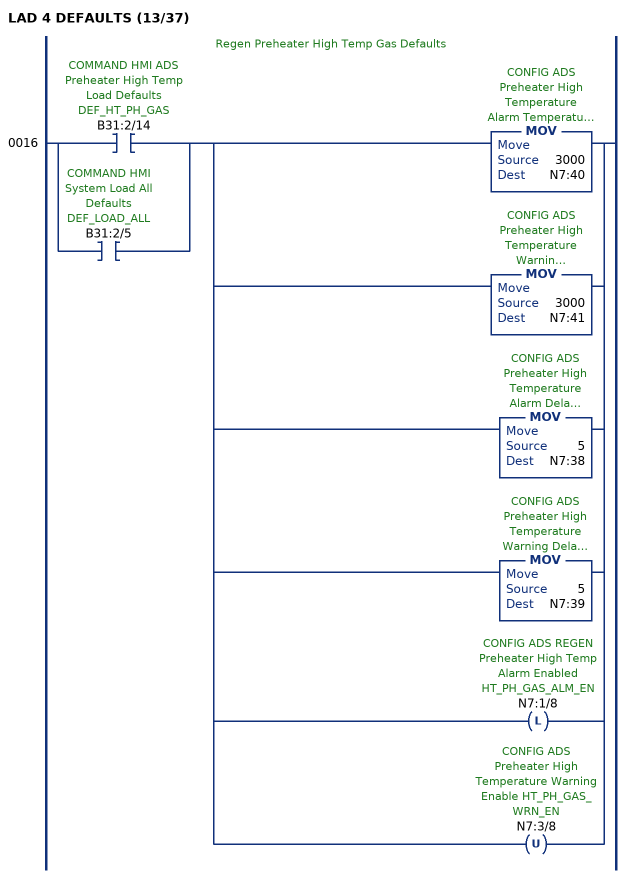
% Rung: 16 %
% Regen Preheater High Temp Gas Defaults %
SOR BST XIC B31:2/14 NXB XIC B31:2/5 BND BST MOV 3000 N7:40 NXB MOV 3000 N7:41 NXB MOV 5 N7:38 NXB MOV 5 N7:39 NXB OTL N7:1/8 NXB OTU N7:3/8 BND EOR
%   B31:2/14  DEF_HT_PH_GAS  "COMMAND HMI ADS Preheater High Temp Load Defaults" %
%   B31:2/5  DEF_LOAD_ALL  "COMMAND HMI System Load All Defaults" %
%   N7:40  HT_PH_GAS_ALM_SP  "CONFIG ADS Preheater High Temperature Alarm Temperature" %
%   N7:41  HT_PH_GAS_WRN_SP  "CONFIG ADS Preheater High Temperature Warning Temperature" %
%   N7:38  HT_PH_GAS_ALM_DLY  "CONFIG ADS Preheater High Temperature Alarm Delay" %
%   N7:39  HT_PH_GAS_WRN_DLY  "CONFIG ADS Preheater High Temperature Warning Delay" %
%   N7:1/8  HT_PH_GAS_ALM_EN  "CONFIG ADS REGEN Preheater High Temp Alarm Enabled" %
%   N7:3/8  HT_PH_GAS_WRN_EN  "CONFIG ADS Preheater High Temperature Warning Enable" %

